{attribute 'qualified_only'}
VAR_GLOBAL
	aRecipe		: ARRAY[1..100] OF RecipeStep; //Recipe Structure
	iRcpTotalStep			: INT; //Recip Total Number
	
	iRcpStepN				: INT;
	cmd_RcpOperation		: INT; // 0:Inital State, 10:RUN, 20:PAUSE, 30:RESTART, 40:STOP, 60:SKIP, 90:ManualOperation
	userState				: INT;	// 0:Inital State, 10:RUN, 20:PAUSE, 30:RESTART, 40:STOP, 50:END, 60:SKIP
	tRecipeControl_Ramp_ET	: TIME;
	tRecipeControl_Hold_ET	: TIME;
	tRecipeControl_Pause_ET	: TIME;
END_VAR

(* stored: Version 1.1.0.1, ProductVersion 3.1.4026.11
   GVL RCP: Id {f007839c-f4b4-44cc-b006-21ad8dc161e6} *)
